
// ===== library: MasterCopy "Flancos" =====

FUNCTION "Flancos" : Void   // FC2, STL
{ S7_Optimized_Access := 'TRUE' }
VERSION : 0.1
BEGIN

REGION Network 1
         A     "ON";
         FP    "M_flanco";
         =     "PON";
END_REGION
END_FUNCTION

// ===== library: MasterCopy "Producción" =====

FUNCTION_BLOCK "Producción"   // FB1, STL
{ S7_Optimized_Access := 'TRUE' }
VERSION : 0.1
BEGIN

REGION Network 1
         A     "X0";
         A     "PON";
         AN    "OFF";

         R     "X0";
         S     "XM1";
   //seguir
END_REGION
END_FUNCTION_BLOCK

// ===== library: MasterCopy "Emergencia" =====

FUNCTION "Emergencia" : Void   // FC3, STL
{ S7_Optimized_Access := 'TRUE' }
VERSION : 0.1
BEGIN

REGION Network 1: Pasar de cualquier estado al estado de emergencia mediante la seta 'EMER'
   // Se establece el estado de defecto "X_EMER" y se resetean el resto de estados.
         A     "EMER";
         S     "X_EMER";

         R     "X0";
         R     "X_ON";
         R     "X_OFF";
         R     "XM1";
         R     "X1";
         R     "XM2";
         R     "X2";
         R     "XM3";
         R     "X3";
         R     "XM4";
         R     "X4";
         R     "XM5";
         R     "X5";
         R     "XM6";
         R     "X6";
         R     "X10";
         R     "X11";
         R     "X12";
END_REGION

REGION Network 2: Tratamiento de X_EMER
   // Se llama a todas las macroetapas, forzando como TRUE el valor de RESET, para que cada macroetapa haga la gestión de la emergencia.
         A     "X_EMER";
         JCN   _TratamientoEmergencia;
   //CALL a todas las macroetapas, metiendolas RESET:= TRUE


   _TratamientoEmergencia:NOP   0;
END_REGION

REGION Network 3: Rearme de la celda mediante el pulsador de rearme sin estar la seta activada.
         A     "X_EMER";
         A     "rearme";
         S     "X0";
         R     "X_EMER";
END_REGION
END_FUNCTION

// ===== library: MasterCopy "maniobra_barnizado" =====

FUNCTION_BLOCK "maniobra_barnizado"   // FB2, STL
{ S7_Optimized_Access := 'TRUE' }
VERSION : 0.1
BEGIN
END_FUNCTION_BLOCK

// ===== library: MasterCopy "test_barnizado" =====

FUNCTION "test_barnizado" : Void   // FC4, STL
{ S7_Optimized_Access := 'TRUE' }
VERSION : 0.1
BEGIN
END_FUNCTION